// TwinCAT 3 PLC project TcTcpUdpRT
// Title: TcTcpUdpRT
// Company: TcInterfaces
// Author: R&B
// ProjectVersion: 1.3.1.0
// ProgramVersion: 3.1.4026.20
// libraries:
//   Tc2_Standard, * (Beckhoff Automation GmbH)
//   Tc2_System, * (Beckhoff Automation GmbH)
//   Tc2_Utilities, * (Beckhoff Automation GmbH)
// project tree:
//   Example/ AppExample.TcPOU, CommunicationExample.TcPOU
//   GVLs/ TcTcpUdpRT_Param.TcGVL
//   ITFs/ IArpPing.TcIO (not stored), ITcpClient.TcIO (not stored), ITcpServer.TcIO (not stored), IUdpSendReceive.TcIO (not stored)
//   POUs/Helper/ IpAddressToLongInt.TcPOU, LongIntToIpAddress.TcPOU (not stored), RingBuffer.TcPOU
//   POUs/ TcArpPing.TcPOU (not stored), TcTcpClient.TcPOU (not stored), TcTcpServer.TcPOU (not stored), TcUdpSendReceive.TcPOU (not stored)
//   Version/ Global_Version.TcGVL

// ---- GVLs/TcTcpUdpRT_Param.TcGVL
{attribute 'qualified_only'}
VAR_GLOBAL CONSTANT
	RingBufferSize		: UDINT := 32768;  // Default ring buffer size for the receivers (32kB). Override per instance with the BufferSize FB_init parameter.
	UdpSourcePortStart	: UINT := 51000;  // Starting range for source port of the UDP instances (51000).
	ErrorStringSize		: UINT := 120;  // Size of error string (120).
	PingRetransmitInterval	: TIME := T#1S;  // Ping resends the echo request at this interval until a reply arrives or the timeout expires (1 s).
END_VAR

// ---- Version/Global_Version.TcGVL
{attribute 'TcGenerated'}
{attribute 'no-analysis'}
{attribute 'linkalways'}
// This function has been automatically generated from the project information.
VAR_GLOBAL CONSTANT
	{attribute 'const_non_replaced'}
	stLibVersion_TcTcpUdpRT : ST_LibVersion := (iMajor := 1, iMinor := 3, iBuild := 1, iRevision := 0, nFlags := 0, sVersion := '1.3.1.0');
END_VAR

// ---- Example/AppExample.TcPOU
PROGRAM AppExample
VAR
	TcServer: TcTcpServer(BufferSize:= 1024);  // Receive buffer size per instance. Initialize the OTCID for the TcServer in the project instance
	Communication: CommunicationExample;
END_VAR

Communication(Server:= TcServer);  // Dependency inject the TcTcpServer implementation into the FB

END_PROGRAM

// ---- Example/CommunicationExample.TcPOU
FUNCTION_BLOCK CommunicationExample
VAR_INPUT
	Server: ITcpServer;
END_VAR
VAR
	iCase: INT;
	rxData: STRING;
	errorMsg: STRING;
END_VAR

// Open and listen for a client on port 9900.
// When client is connected, receive data until 'disconnect' command it received.

Server.Run();  // Must be called cyclic to maintain the communication between the PLC code and the IO.

CASE iCase OF 
	0:
		IF Server.OpenConnection(9900) THEN
			iCase := iCase + 1;
		END_IF
	1:
		IF Server.IsConnected THEN
			iCase := iCase + 1;
		END_IF
	2:
		IF Server.IsDataAvailable THEN
			Server.Receive(DataPointer:= ADR(rxData), DataLength:= SIZEOF(rxData));
			IF rxData = 'disconnect' THEN
				iCase:= iCase + 1;
			END_IF
		END_IF
	3:
		IF Server.CloseConnection() THEN
			iCase := 0;
		END_IF
END_CASE

IF Server.Error THEN
	errorMsg := Server.GetError;
	iCase := -1;
END_IF

END_FUNCTION_BLOCK

// ---- POUs/Helper/IpAddressToLongInt.TcPOU
// Format the string IP address to a long integer value.
// '192.168.17.10' => 0xC0A8110A
FUNCTION IpAddressToLongInt : UDINT
VAR_INPUT
	IpAddress: STRING(15);
END_VAR
VAR
	i: UINT;
	pos: INT;
	value : UDINT;
END_VAR

FOR i := 0 TO 3 DO
	IpAddressToLongInt := ROL(IpAddressToLongInt, 8);
	IF i < 3 THEN
		pos := FIND(STR1:= IpAddress, STR2:= '.');
		value := STRING_TO_UDINT(LEFT(IpAddress, pos-1));
	ELSE
		value := STRING_TO_UDINT(IpAddress);
	END_IF
	IpAddressToLongInt := IpAddressToLongInt OR value;
	IpAddress := DELETE(STR:= IpAddress, LEN:= pos, POS:= 1);
END_FOR

END_FUNCTION

// ---- POUs/Helper/RingBuffer.TcPOU
// The buffer uses 1-byte separation rule from the writer to the reader.
// The storage is allocated once from the TwinCAT router memory with __NEW in Init()
// and released again with __DELETE in FB_exit. Call Init() during start-up (e.g. from
// the FB_init of the owning function block) before using the buffer.
FUNCTION_BLOCK RingBuffer
VAR
	_error			: BOOL;
	_errorString	: STRING(TcTcpUdpRT_Param.ErrorStringSize);
	_pBuffer		: POINTER TO BYTE;  // Dynamically allocated storage (__NEW), 0 when not allocated
	_size			: UDINT;  // Size of the allocated storage in bytes
	_readPointer	: UDINT;
	_writePointer	: UDINT;
END_VAR

METHOD PRIVATE CopyFromBuffer : UDINT
VAR_INPUT
	Data	: POINTER TO BYTE;
	Length	: UDINT;
END_VAR
CopyFromBuffer := MEMCPY(destAddr:= Data, srcAddr:= ADR(_pBuffer[_readPointer]), n:= Length);
IF CopyFromBuffer = 0 THEN
	_error := TRUE;
	_errorString := CONCAT('MEMCPY invalid parameter, ReadPointer: ', CONCAT(TO_STRING(_readPointer), CONCAT(', Length: ', CONCAT(TO_STRING(Length), CONCAT(', Data: ', TO_STRING(Data))))));
ELSIF CopyFromBuffer <> Length THEN
	_error := TRUE;
	_errorString := CONCAT('MEMCPY size ', CONCAT(TO_STRING(CopyFromBuffer), CONCAT(' from buffer is different from length ', TO_STRING(Length))));
ELSE
	_readPointer := (_readPointer + CopyFromBuffer) MOD _size;
END_IF
END_METHOD

METHOD PRIVATE CopyToBuffer : UDINT
VAR_INPUT
	Data	: POINTER TO BYTE;
	Length	: UDINT;
END_VAR
CopyToBuffer := MEMCPY(destAddr:= ADR(_pBuffer[_writePointer]), srcAddr:= Data, n:= Length);
IF CopyToBuffer = 0 THEN
	_error := TRUE;
	_errorString := CONCAT('MEMCPY invalid parameter, WritePointer: ', CONCAT(TO_STRING(_writePointer), CONCAT(', Length: ', CONCAT(TO_STRING(Length), CONCAT(', Data: ', TO_STRING(Data))))));
ELSIF CopyToBuffer <> Length THEN
	_error := TRUE;
	_errorString := CONCAT('MEMCPY size ', CONCAT(TO_STRING(CopyToBuffer), CONCAT(' to buffer is different from length ', TO_STRING(Length))));
ELSE
	_writePointer := (_writePointer + CopyToBuffer) MOD _size;
END_IF
END_METHOD

METHOD EmptyBuffer : BOOL
VAR
	set	: UDINT;
END_VAR
IF _pBuffer = 0 THEN
	_error := TRUE;
	_errorString := 'Ring buffer is not allocated, call Init() first';
	RETURN;
END_IF

set := MEMSET(destAddr:= _pBuffer, fillByte:= 0, n:= _size);
IF set = _size THEN
	_readPointer := 0;
	_writePointer := 0;
	EmptyBuffer := TRUE;
ELSE
	_error := TRUE;
	_errorString := 'Failed to empty ring buffer, MEMSET to zero';
END_IF
END_METHOD

PROPERTY Error : BOOL
GET
Error := _error;
END_GET
END_PROPERTY

//FB_Exit must be implemented explicitly. If there is an implementation, then the
//method is called before the controller removes the code of the function block instance
//(implicit call). The return value is not evaluated.
METHOD FB_Exit: BOOL
VAR_INPUT
    bInCopyCode: BOOL;  // TRUE: the exit method is called in order to leave the instance which will be copied afterwards (online change).  
END_VAR
IF NOT bInCopyCode AND _pBuffer <> 0 THEN  // No online change -> shutdown, release the router memory
	__DELETE(_pBuffer);  // Sets _pBuffer to 0
	_size := 0;
END_IF
END_METHOD

PROPERTY GetError : STRING(TcTcpUdpRT_Param.ErrorStringSize)
GET
GetError := _errorString;
END_GET
END_PROPERTY

METHOD Init : BOOL
VAR_INPUT
	BufferSize	: UDINT;  // Size of the ring buffer in bytes, 0 uses TcpUdp_Param.RingBufferSize
END_VAR
IF _pBuffer <> 0 THEN
	Init := TRUE;  // Already allocated, allocation is only done once
	RETURN;
END_IF

IF BufferSize = 0 THEN
	BufferSize := TcTcpUdpRT_Param.RingBufferSize;
END_IF

_pBuffer := __NEW(BYTE, BufferSize);
IF _pBuffer = 0 THEN
	_size := 0;
	_error := TRUE;
	_errorString := CONCAT('Failed to allocate ring buffer of size ', CONCAT(TO_STRING(BufferSize), ' from router memory'));
	RETURN;
END_IF

_size := BufferSize;
_readPointer := 0;
_writePointer := 0;
Init := TRUE;
END_METHOD

PROPERTY IsAllocated : BOOL
GET
IsAllocated := _pBuffer <> 0;
END_GET
END_PROPERTY

PROPERTY IsBufferEmpty : BOOL
GET
IF _size = 0 THEN
	IsBufferEmpty := TRUE;
	RETURN;
END_IF
IsBufferEmpty := (TO_LINT((_readPointer - _writePointer + _size) MOD _size) - 1) = -1;
END_GET
END_PROPERTY

PROPERTY IsBufferFull : BOOL
GET
IF _size = 0 THEN
	IsBufferFull := FALSE;
	RETURN;
END_IF
IsBufferFull := (TO_LINT((_readPointer - _writePointer + _size) MOD _size) - 1) = 0;
END_GET
END_PROPERTY

METHOD Read : UDINT
VAR_INPUT
	Data	: POINTER TO BYTE;
	Length	: UDINT;
END_VAR
VAR
	copied	: UDINT;
	first	: UDINT;
	second	: UDINT;
	available	: UDINT;
END_VAR
IF _pBuffer = 0 THEN
	_error := TRUE;
	_errorString := 'Ring buffer is not allocated, call Init() first';
	RETURN;
ELSIF Data = 0 THEN
	Read := 0;
	_error := TRUE;
	_errorString := 'Was not able to read from buffer because data pointer was empty';
	RETURN;
ELSIF Length = 0 THEN
	Read := 0;
	_error := TRUE;
	_errorString := 'Was not able to read from buffer because length was zero';
	RETURN;
END_IF

IF _readPointer = _writePointer THEN
	// No data to be read
    Read := 0;
    RETURN;
END_IF

available := (_writePointer - _readPointer + _size) MOD _size;
IF Length > available THEN
	// Only read available data
	Length := available;
END_IF

IF _readPointer + Length <= _size THEN
	// No wrap around
	Read := CopyFromBuffer(Data:= Data, Length:= Length);
ELSE
	// Wrap around
	first := _size - _readPointer;
	copied := CopyFromBuffer(Data:= Data, Length:= first);
	Read := copied;
	
	IF _error THEN
		RETURN;
	END_IF
	
	second := Length - first;
	copied := CopyFromBuffer(Data:= ADR(Data[first]), Length:= second);
	Read := Read + copied;
END_IF
END_METHOD

METHOD ResetError
_error := FALSE;
_errorString := '';
END_METHOD

PROPERTY Size : UDINT
GET
Size := _size;
END_GET
END_PROPERTY

METHOD Write : UDINT
VAR_INPUT
	Data	: POINTER TO BYTE;
	Length	: UDINT;
END_VAR
VAR
	copied	: UDINT;
	first	: UDINT;
	second	: UDINT;
	available	: LINT;
END_VAR
IF _pBuffer = 0 THEN
	_error := TRUE;
	_errorString := 'Ring buffer is not allocated, call Init() first';
	RETURN;
ELSIF Data = 0 THEN
	Write := 0;
	_error := TRUE;
	_errorString := 'Was not able to write to buffer because data pointer was empty';
	RETURN;
ELSIF Length = 0 THEN
	Write := 0;
	_error := TRUE;
	_errorString := 'Was not able to write to buffer because length was zero';
	RETURN;
END_IF

IF IsBufferEmpty THEN
	available := _size - 1;
ELSE
	available := TO_LINT((_readPointer - _writePointer + _size) MOD _size) - 1;
END_IF

IF Length > available THEN 
	// Not enough space available
	Write := 0;
	_error := TRUE;
	_errorString := CONCAT('Ring buffer write overflow, available: ', CONCAT(TO_STRING(available), CONCAT(', length: ', TO_STRING(Length))));
	RETURN;
END_IF

IF (_writePointer + Length) <= _size THEN
	// No wrap around
	Write := CopyToBuffer(Data:= Data, Length:= Length);
ELSE
	// Wrap around
	first := _size - _writePointer;
	copied := CopyToBuffer(Data:= Data, Length:= first);
	Write := copied;
	
	IF _error THEN
		RETURN;
	END_IF
	
	second := Length - first;
	copied := CopyToBuffer(Data:= ADR(Data[first]), Length:= second);
	Write := Write + copied;
END_IF
END_METHOD

END_FUNCTION_BLOCK
